(* IEC 61131-3 sources: POMIRTS_lab3/AS/Library_2/MTWinder/V1.00.3, 3 files *)

(* ---- MTWinder.typ ---- *)
TYPE
	MTWinderAxisControllerIntType : 	STRUCT  (*Data for internal use.*)
		CycleTime : REAL; (*Task cycle time. Unit: [s].*)
		Configuration : MTWinderConfigurationType; (*Data for internal use.*)
		Parameters : MTWinderAxisControllerType; (*Data for internal use.*)
		ParametersValid : BOOL; (*Data for internal use.*)
		UpdateOld : BOOL; (*Data for internal use.*)
		StartSynchronizationOld : BOOL; (*Data for internal use.*)
		StopSynchronizationOld : BOOL; (*Data for internal use.*)
		EnableOld : BOOL; (*Data for internal use.*)
		Update : BOOL; (*Data for internal use.*)
		WinderRatio : LREAL; (*Data for internal use.*)
		ActualDiameter : REAL; (*Data for internal use.*)
		ActIntegrationTime : REAL; (*Data for internal use.*)
		ActProportionalGainOld : REAL; (*Data for internal use.*)
		ActProportionalGain : REAL; (*Data for internal use.*)
		ActualInertia : REAL; (*Data for internal use.*)
		RollerDensity : REAL; (*Data for internal use.*)
		StatusIDUpdate : DINT; (*Data for internal use.*)
		StatusIDCommando : DINT; (*Data for internal use.*)
		StatusIDCyclic : DINT; (*Data for internal use.*)
		InSynchronizationOld : BOOL; (*Data for internal use.*)
		SynchronizationParameters : MTWinderAxisControllerSyncType; (*Data for internal use.*)
		SetLineVelocitySampled : REAL; (*Data for internal use.*)
	END_STRUCT;
	MTWinderAxisControllerSyncEnum :
		( (*Synchronization state of the axis controller.*)
		mtWND_STATE_STOP := 0, (*Data for internal use.*)
		mtWND_STATE_RAMP_UP := 1, (*Data for internal use.*)
		mtWND_STATE_IN_SYNC := 2, (*Data for internal use.*)
		mtWND_STATE_RAMP_DOWN := 3 (*Data for internal use.*)
		);
	MTWinderAxisControllerSyncType : 	STRUCT  (*Ramp up time parameters for the synchronization.*)
		SyncState : MTWinderAxisControllerSyncEnum; (*Data for internal use.*)
		SyncLineVelocity : REAL; (*Data for internal use.*)
		SyncLineVelocityOld : REAL; (*Data for internal use.*)
		SyncLineAcceleration : REAL; (*Data for internal use.*)
		alpha : REAL; (*Data for internal use.*)
		SyncTime : REAL; (*Data for internal use.*)
	END_STRUCT;
	MTWinderAxisControllerType : 	STRUCT  (*Parameter for the winder axis.*)
		MinTorque : REAL; (*Lower limit for the motor torque preset value SetMotorTorque. Unit: [Nm]. *)
		MaxTorque : REAL; (*Upper limit for the motor torque preset value SetMotorTorque. Unit: [Nm].*)
		Interpolation : MTWinderInterpolationType; (*Parameter for interpolating the speed controller parameters of the winder axis.*)
	END_STRUCT;
	MTWinderAxisType : 	STRUCT  (*Axis parameter.*)
		LineUnits : REAL; (*Scaling of the line position. Unit: [Units/m]. *)
		WinderUnits : UDINT; (*Scaling of the winder axis. Unit: [Units].*)
		RevMotor : UDINT; (*Number of motor revolutions required for the position of the winder to increase/decrease by a number of units equal to WinderUnits. Unit: [Rev]. *)
		GearRatio : REAL; (*Gear ratio between the motor and winder (motor speed ÷ winder speed). Unit: [1]. *)
		WinderType : MTWinderTypeEnum; (*Selects whether the system is a winder or unwinder unit.*)
		ReverseWinderDirection : BOOL; (*Changes the direction of rotation for the winder axis.*)
	END_STRUCT;
	MTWinderConfigurationType : 	STRUCT  (*Configuration parameters for the winder and the motor.*)
		Geometry : MTWinderGeometryType; (*Geometric parameter of winder.*)
		Axis : MTWinderAxisType; (*Axis parameter.*)
	END_STRUCT;
	MTWinderControllerType : 	STRUCT  (*Parameter for setting the controller.*)
		PIDParameters : MTPIDParametersType; (*PID parameter.*)
		MaxLineVelocityCorrection : REAL; (*Maximum permitted correction by controller depending on the line velocity. Unit: [mm/s].*)
		MaxControlError : REAL; (*Threshold value for detecting material failure. Unit: [mm] for closed-loop dancer control, [N] for closed-loop tension control.*)
	END_STRUCT;
	MTWinderDancerControllerIntType : 	STRUCT  (*Data for internal use.*)
		CycleTime : REAL; (*Task cycle time. Unit: [s].*)
		Configuration : MTWinderConfigurationType; (*Data for internal use.*)
		Parameters : MTWinderControllerType; (*Data for internal use.*)
		ParametersValid : BOOL; (*Data for internal use.*)
		UpdateOld : BOOL; (*Data for internal use.*)
		EnableOld : BOOL; (*Data for internal use.*)
		WinderRatio : LREAL; (*Data for internal use.*)
		ActualDiameter : REAL; (*Data for internal use.*)
		MaterialBreak : BOOL; (*Data for internal use.*)
		ControlError : REAL; (*Data for internal use.*)
		ControlErrorOld : REAL; (*Data for internal use.*)
		PIDStatusID : DINT; (*Data for internal use.*)
		ProportionalPart : REAL; (*Data for internal use.*)
		IntegrationPart : REAL; (*Data for internal use.*)
		DerivativePart : REAL; (*Data for internal use.*)
		ControllerOutput : REAL; (*Data for internal use.*)
		HoldIntegration : MTPIDIntegrationEnum; (*Data for internal use.*)
		IntegrationStatus : MTPIDIntegrationEnum; (*Data for internal use.*)
		StatusIDUpdate : DINT; (*Data for internal use.*)
	END_STRUCT;
	MTWinderDiameterEstBufferParType : 	STRUCT  (*Buffer parameters for the diameter estimator.*)
		Counter : USINT; (*Data for internal use.*)
		Index : USINT; (*Data for internal use.*)
		ActDiameter : ARRAY[0..99]OF LREAL; (*Data for internal use.*)
		WinderRevolution : ARRAY[0..99]OF LREAL; (*Data for internal use.*)
	END_STRUCT;
	MTWinderDiameterEstInternalType : 	STRUCT  (*Data for internal use.*)
		CycleTime : REAL; (*Task cycle time. Unit: [s].*)
		Configuration : MTWinderConfigurationType; (*Data for internal use.*)
		Parameters : MTWinderDiameterEstType; (*Data for internal use.*)
		ParametersValid : BOOL; (*Data for internal use.*)
		UpdateOld : BOOL; (*Data for internal use.*)
		EnableOld : BOOL; (*Data for internal use.*)
		Mode : MTWinderDiameterEstModeEnum; (*Data for internal use.*)
		SetPresetDiameterOld : BOOL; (*Data for internal use.*)
		PresetDiameter : REAL; (*Data for internal use.*)
		WinderRatio : LREAL; (*Data for internal use.*)
		RollerDensity : REAL; (*Data for internal use.*)
		SetPresetDiameterMode : USINT; (*Data for internal use.*)
		ReverseWinder : SINT; (*Data for internal use.*)
		MaterialBreak : BOOL; (*Data for internal use.*)
		SystemParameters : MTWinderDiameterEstSysParType; (*Data for internal use.*)
		EstimationParameters : MTWinderDiameterEstParType; (*Data for internal use.*)
		BufferParameters : MTWinderDiameterEstBufferParType; (*Data for internal use.*)
		LQFilter : MTWinderDiameterEstLQFilterType; (*Data for internal use.*)
		ActDiameter : REAL; (*Data for internal use.*)
		AvgMaterialThickness : REAL; (*Data for internal use.*)
		MinDiameterAchieved : BOOL; (*Data for internal use.*)
		ActLinePosition : DINT; (*Data for internal use.*)
		ActLinePositionOld : DINT; (*Data for internal use.*)
		FilterWindowTime : LREAL; (*Data for internal use.*)
		RemainingRunTime : ARRAY[0..2]OF REAL; (*Data for internal use.*)
		LineVelocity : REAL; (*Data for internal use.*)
	END_STRUCT;
	MTWinderDiameterEstLQFilterType : 	STRUCT  (*Filter parameters for the diameter estimator.*)
		LQError : REAL; (*Data for internal use.*)
		LQOutputFiltered : ARRAY[0..1]OF LREAL; (*Data for internal use.*)
		LQOutput : ARRAY[0..1]OF REAL; (*Data for internal use.*)
		LQParameterVector : ARRAY[0..2]OF REAL; (*Data for internal use.*)
		UpdateFilter : BOOL; (*Data for internal use.*)
		ResetFilter : BOOL; (*Data for internal use.*)
		InitFilter : BOOL; (*Data for internal use.*)
		NumberOfDataVector : UDINT; (*Data for internal use.*)
		BVector : ARRAY[0..1]OF DINT; (*Data for internal use.*)
		XVector : ARRAY[0..1]OF LREAL; (*Data for internal use.*)
	END_STRUCT;
	MTWinderDiameterEstModeEnum :
		( (*Diameter estimation mode.*)
		mtWND_NO_ESTIMATION := 0, (*Disables the diameter estimation.*)
		mtWND_POSITION_BASED := 1, (*Cyclic diameter estimation based on differences in position.*)
		mtWND_VELOCITY_INTEGRATION_BASED := 2 (*Cyclic diameter estimation based on integrated speeds.*)
		);
	MTWinderDiameterEstParType : 	STRUCT  (*Estimation parameters for the diameter estimator.*)
		ActDiameter : LREAL; (*Data for internal use.*)
		ActDiameterOld : REAL; (*Data for internal use.*)
		ActDiameterCorrect : REAL; (*Data for internal use.*)
		ActDiameterStart : REAL; (*Data for internal use.*)
		StartEstimation : BOOL; (*Data for internal use.*)
		StartLinePosition : DINT; (*Data for internal use.*)
		StartWinderPosition : DINT; (*Data for internal use.*)
		StartDancerPosition : REAL; (*Data for internal use.*)
		LinePositionIntegration : LREAL; (*Data for internal use.*)
		WinderPositionIntegration : LREAL; (*Data for internal use.*)
		ActWinderRevolution : ARRAY[0..2]OF LREAL; (*Data for internal use.*)
		WinderRevolution : LREAL; (*Data for internal use.*)
		ActLinePositionOld : DINT; (*Data for internal use.*)
	END_STRUCT;
	MTWinderDiameterEstSysParType : 	STRUCT  (*System parameters for the diameter estimator.*)
		ActWinderPositionOld : DINT; (*Data for internal use.*)
		ActWinderPositionDelta : DINT; (*Data for internal use.*)
		ActWinderRevolution : LREAL; (*Data for internal use.*)
		ActMotorRevolution : ARRAY[0..1]OF UDINT; (*Data for internal use.*)
	END_STRUCT;
	MTWinderDiameterEstType : 	STRUCT  (*Parameter for diameter estimation.*)
		CyclicEstimationWindow : UDINT; (*Duration of the cyclic estimation window for estimating the diameter. Unit: [Units].*)
		FilterWindow : UDINT; (*Position-related filter constant for the filter. Unit: [Units].*)
		MaterialBreakThreshold : REAL; (*Window for detecting material failure. Unit: [mm].*)
	END_STRUCT;
	MTWinderGeometryType : 	STRUCT  (*Geometric parameter of winder.*)
		WinderWidth : REAL; (*Width of the winder. Unit: [mm]. *)
		MaterialThickness : REAL; (*Material thickness or diameter (e.g. of the wire). Unit: [µm]. *)
		MaxDiameter : REAL; (*Maximum winder diameter. Unit: [mm]. *)
		MinDiameter : REAL; (*Minimum winder diameter. Unit: [mm].*)
		MinInertia : REAL; (*Moment of inertia of the winder at diameter MinDiameter. Unit: [kgm˛]. *)
		TestDiameter : REAL; (*Winder diameter between the minimum and maximum diameter at which the TestInertia or TestProportionalGain and TestIntegrationTime are determined. This diameter should be as large as possible. Unit: [mm].*)
		TestInertia : REAL; (*Moment of inertia of the winder at diameter TestDiameter. Unit: [kgm˛]. *)
	END_STRUCT;
	MTWinderInterpolationType : 	STRUCT  (*Parameter for interpolating the speed controller parameters of the winder axis.*)
		MinProportionalGain : REAL; (*Proportional gain of speed controller at minimum diameter MinDiameter. Unit: [As].*)
		TestProportionalGain : REAL; (*Proportional gain of speed controller at diameter TestDiameter. Unit: [As].*)
		MinIntegrationTime : REAL; (*Integration time of speed controller at minimum diameter. Unit: [s].*)
		TestIntegrationTime : REAL; (*Integration time of speed controller at diameter TestDiameter. Unit: [s].*)
	END_STRUCT;
	MTWinderModelTypeEnum :
		( (*Model for the winder application.*)
		mtWND_DANCER := 0, (*Uses the simulation model for dancer control.*)
		mtWND_TENSION_CLOSED_LOOP := 1, (*Uses the simulation model for closed-loop tension control.*)
		mtWND_TENSION_OPEN_LOOP := 2 (*Uses the simulation model for open-loop tension control.*)
		);
	MTWinderSimMaterialParType : 	STRUCT  (*Simulation model material parameters.*)
		RollerDensity : REAL; (*Roller density [kg/mł].*)
		ElasticityConstant : REAL; (*Elacticity constant [N/mm˛].*)
		Elongation : REAL; (*Elongation [N/m˛].*)
		Material : USINT; (*Plastic = 0. Paper = 1.*)
	END_STRUCT;
	MTWinderSimSystemParType : 	STRUCT  (*Simulation model system parameters.*)
		LinePosition : LREAL; (*Actual line position, [m]*)
		LineVelocity : LREAL; (*Actual line velocity, [m/s]*)
		IntegratorState : LREAL; (*Integrator state.*)
		MaterialTension : ARRAY[0..2]OF LREAL; (*Material tension [N].*)
		DancerArmPosition : ARRAY[0..2]OF LREAL; (*Dancer arm position [rad].*)
		DancerArmVelocity : ARRAY[0..2]OF LREAL; (*Dancer arm velocity [rad/s].*)
		WinderRollerPosition : ARRAY[0..2]OF LREAL; (*Winder roller position [rad].*)
		WinderRollerVelocity : ARRAY[0..2]OF LREAL; (*Winder roller velocity [rad/s].*)
		UnwoundMaterialLength : ARRAY[0..2]OF LREAL; (*Unwound material length [mm].*)
	END_STRUCT;
	MTWinderSimulationModelIntType : 	STRUCT  (*Data for internal use.*)
		CycleTime : REAL; (*Task cycle time. Unit: [s].*)
		Configuration : MTWinderConfigurationType; (*Data for internal use.*)
		Parameters : MTWinderSimulationModelType; (*Data for internal use.*)
		SystemParameters : MTWinderSimSystemParType; (*Data for internal use.*)
		MaterialParameters : MTWinderSimMaterialParType; (*Data for internal use.*)
		ParametersValid : BOOL; (*Data for internal use.*)
		UpdateOld : BOOL; (*Data for internal use.*)
		EnableOld : BOOL; (*Data for internal use.*)
		ActualDiameter : REAL; (*Data for internal use.*)
		InitSpeedControllerOld : REAL; (*Data for internal use.*)
		ActProportionalGain : REAL; (*Data for internal use.*)
		ActIntegrationTime : REAL; (*Data for internal use.*)
		MaterialBreak : BOOL; (*Data for internal use.*)
		ModelType : MTWinderModelTypeEnum; (*Data for internal use.*)
		TorqueMode : MTWinderTorqueModeEnum; (*Data for internal use.*)
		Update : BOOL; (*Data for internal use.*)
		InhibitUpdate : BOOL; (*Data for internal use.*)
	END_STRUCT;
	MTWinderSimulationModelType : 	STRUCT  (*Parameter for the simulation model.*)
		MaterialLength : REAL; (*Material length between the unwinder and infeed or between the outfeed and winder. Unit: [mm]. *)
		StartDiameter : REAL; (*Winder diameter used to start the simulation. Unit: [mm]. *)
		MaxDancerPosition : REAL; (*Maximum position of the dancer arm. Unit: [mm]. *)
		DancerLength : REAL; (*Length of the dancer arm. Unit: [mm]. *)
		DancerInertia : REAL; (*Moment of inertia of the dancer. Unit: [kgm˛]. *)
		SpeedTorqueFactor : REAL; (*Friction coefficient for the winder proportional to the velocity. Unit: [Nms]. *)
		TorqueConstant : REAL; (*Torque constant of the motor from the winder Unit: [Nm/A]. *)
		Noise : BOOL; (*Enables noise for the ActLinePosition, ActLineVelocity, ActWinderPosition, ActWinderVelocity, ActDancerPosition and ActMaterialTension outputs.*)
	END_STRUCT;
	MTWinderTaperTensionInternalType : 	STRUCT  (*Data for internal use.*)
		CycleTime : REAL; (*Task cycle time. Unit: [s].*)
		Configuration : MTWinderConfigurationType; (*Data for internal use.*)
		Parameters : MTWinderTaperTensionType; (*Data for internal use.*)
		ParametersValid : BOOL; (*Data for internal use.*)
		UpdateOld : BOOL; (*Data for internal use.*)
		EnableOld : BOOL; (*Data for internal use.*)
		ActualDiameter : REAL; (*Data for internal use.*)
		StartMotorTorque : REAL; (*Data for internal use.*)
		MaxMotorTorque : REAL; (*Data for internal use.*)
		MinMotorTorque : REAL; (*Data for internal use.*)
		SetMotorTorque : REAL; (*Data for internal use.*)
		StatusIDUpdate : DINT; (*Data for internal use.*)
	END_STRUCT;
	MTWinderTaperTensionModeEnum :
		( (*Tension curve mode.*)
		mtWND_LINEAR_DECREASE_TENSION := 0, (*Linear reduction of the tension.*)
		mtWND_LINEAR_DECREASE_TORQUE := 1 (*Linear reduction of the torque.*)
		);
	MTWinderTaperTensionType : 	STRUCT  (*Parameter for determining the tension profile.*)
		StartDiameter : REAL; (*Tension is reduced beginning with this diameter. Unit: [mm].*)
		MaxMaterialTension : REAL; (*Maximum tension. Unit: [N].*)
		MinMaterialTension : REAL; (*Minimum tension. Unit: [N].*)
		Mode : MTWinderTaperTensionModeEnum; (*Tension curve mode.*)
	END_STRUCT;
	MTWinderTensionControllerIntType : 	STRUCT  (*Data for internal use.*)
		CycleTime : REAL; (*Task cycle time. Unit: [s].*)
		Configuration : MTWinderConfigurationType; (*Data for internal use.*)
		Parameters : MTWinderControllerType; (*Data for internal use.*)
		ParametersValid : BOOL; (*Data for internal use.*)
		UpdateOld : BOOL; (*Data for internal use.*)
		EnableOld : BOOL; (*Data for internal use.*)
		WinderRatio : LREAL; (*Data for internal use.*)
		ActualDiameter : REAL; (*Data for internal use.*)
		MaterialBreak : BOOL; (*Data for internal use.*)
		ControlError : REAL; (*Data for internal use.*)
		ControlErrorOld : REAL; (*Data for internal use.*)
		PIDStatusID : DINT; (*Data for internal use.*)
		ProportionalPart : REAL; (*Data for internal use.*)
		IntegrationPart : REAL; (*Data for internal use.*)
		DerivativePart : REAL; (*Data for internal use.*)
		ControllerOutput : REAL; (*Data for internal use.*)
		HoldIntegration : MTPIDIntegrationEnum; (*Data for internal use.*)
		IntegrationStatus : MTPIDIntegrationEnum; (*Data for internal use.*)
		StatusIDUpdate : DINT; (*Data for internal use.*)
	END_STRUCT;
	MTWinderTorqueModeEnum :
		( (*Specifies how the value of the SetMotorTorque input is used.*)
		mtWND_TORQUE_LIMIT := 40, (*Uses SetMotorTorque for torque limiting.*)
		mtWND_TORQUE_FF := 32 (*Uses SetMotorTorque for feed-forward torque control.*)
		);
	MTWinderTypeEnum :
		( (*Selects whether the system is a winder or unwinder unit.*)
		mtWND_REWIND := -1, (*Winder used for winding.*)
		mtWND_UNWIND := +1 (*Winder used for unwinding.*)
		);
END_TYPE

(* ---- MTWinder.var ---- *)
(*Errors: Common*)
VAR CONSTANT
	mtWND_ERR_GEO_PAR_INVALID : DINT := -1058007184; (*Geometric parameter set for winder is invalid.*)
	mtWND_ERR_AXIS_PAR_INVALID : DINT := -1058007183; (*Axis parameter set for winder is invalid.*)
	mtWND_ERR_MATERIAL_BREAK : DINT := -1058007181; (*Material breakage detected.*)
	mtWND_ERR_ACT_DIAMETER_INVALID : DINT := -1058007167; (*Actual diameter for winder is invalid.*)
END_VAR
(*Warnings: Common*)
VAR CONSTANT
	mtWND_WRN_GEO_PAR_INVALID : DINT := -2131749008; (*Geometric parameter set for winder is invalid.*)
	mtWND_WRN_AXIS_PAR_INVALID : DINT := -2131749007; (*Axis parameter set for winder is invalid.*)
	mtWND_WRN_ACT_DIAMETER_INVALID : DINT := -2131748994; (*Actual diameter for winder is invalid.*)
END_VAR
(*Errors: MTWinderAxisController*)
VAR CONSTANT
	mtWND_ERR_TORQUE_LIMITS_INVALID : DINT := -1058007173; (*Torque limits set for winder are invalid.*)
	mtWND_ERR_INTERPOL_PAR_INVALID : DINT := -1058007172; (*Interpolation parameters are invalid.*)
	mtWND_ERR_SET_MAT_TENSION_NEG : DINT := -1058007169; (*Set material tension is negative.*)
END_VAR
(*Warnings: MTWinderAxisController*)
VAR CONSTANT
	mtWND_WRN_TORQUE_LIMITS_INVALID : DINT := -2131749001; (*Torque limits set for winder are invalid.*)
	mtWND_WRN_INTERPOL_PAR_INVALID : DINT := -2131749000; (*Interpolation parameters are invalid.*)
	mtWND_WRN_SYNC_TIME_NEGATIVE : DINT := -2131748996; (*Synchronization time for winder is invalid.*)
END_VAR
(*Errors: MTWinderDancerController and MTWinderTensionController*)
VAR CONSTANT
	mtWND_ERR_MAX_CONTROL_ERROR_NEG : DINT := -1058007176; (*Max control error for material detection is negative.*)
	mtWND_ERR_LINE_VEL_CORRECTION : DINT := -1058007166; (*Maximum line velocity correction is negative or equal to 0.*)
END_VAR
(*Warnings: MTWinderDancerController and MTWinderTensionController*)
VAR CONSTANT
	mtWND_WRN_MAX_CONTROL_ERROR_NEG : DINT := -2131749004; (*Max control error for material detection is negative.*)
	mtWND_WRN_LINE_VEL_CORRECTION : DINT := -2131748993; (*Maximum line velocity correction is negative or equal to 0.*)
END_VAR
(*Errors: MTWinderDiameterEstimator*)
VAR CONSTANT
	mtWND_ERR_DIAMETER_EST_MODE : DINT := -1058007177; (*Mode for the diameter estimator is invalid.*)
	mtWND_ERR_CYCLIC_EST_WINDOW : DINT := -1058007175; (*Cyclic estimation window for the diameter estimation is invalid.*)
	mtWND_ERR_MAT_BREAK_THRESHOLD : DINT := -1058007168; (*Threshold for material break detection is invalid.*)
END_VAR
(*Warnings: MTWinderDiameterEstimator*)
VAR CONSTANT
	mtWND_WRN_DIAMETER_EST_MODE : DINT := -2131749005; (*Mode for the diameter estimator is invalid.*)
	mtWND_WRN_CYCLIC_EST_WINDOW : DINT := -2131749003; (*Cyclic estimation window for the diameter estimator is invalid.*)
	mtWND_WRN_MIN_DIAMETER_REACHED : DINT := -2131749002; (*The diameter estimator has reached the minimum diameter.*)
	mtWND_WRN_MAT_BREAK_THRESHOLD : DINT := -2131748995; (*Threshold for material break detection is invalid.*)
	mtWND_WRN_PRESET_DIAMETER : DINT := -2131748990; (*Preset diameter for the diameter estimator is invalid.*)
END_VAR
(*Errors: MTWinderSimulationModel*)
VAR CONSTANT
	mtWND_ERR_SIM_PAR_INVALID : DINT := -1058007182; (*Simulation parameter set for winder is invalid.*)
	mtWND_ERR_MODEL_TYPE_INVALID : DINT := -1058007180; (*Type of model is invalid.*)
	mtWND_ERR_TORQUE_MODE_INVALID : DINT := -1058007179; (*Torque mode of model is invalid.*)
	mtWND_ERR_MODEL_TORQUE_INVALID : DINT := -1058007178; (*Torque mode for selected model type is invalid.*)
END_VAR
(*Warnings: MTWinderSimulationModel*)
VAR CONSTANT
	mtWND_WRN_SIM_PAR_INVALID : DINT := -2131749006; (*Simulation parameter set for winder is invalid.*)
END_VAR
(*Errors: MTWinderTaperTension*)
VAR CONSTANT
	mtWND_ERR_START_DIAMETER_INVALID : DINT := -1058007171; (*Start diameter for winder is invalid.*)
	mtWND_ERR_MATERIAL_TENSION_LIMIT : DINT := -1058007165; (*The maximum and the minimum material tension is invalid.*)
	mtWND_ERR_TAPER_TENSION_MODE : DINT := -1058007164; (*Mode for the taper tension is invalid.*)
END_VAR
(*Warnings: MTWinderTaperTension*)
VAR CONSTANT
	mtWND_WRN_START_DIAMETER_INVALID : DINT := -2131748999; (*Start diameter for winder is invalid.*)
	mtWND_WRN_MATERIAL_TENSION_LIMIT : DINT := -2131748992; (*The maximum and the minimum material tension is invalid.*)
	mtWND_WRN_TAPER_TENSION_MODE : DINT := -2131748991; (*Mode for the taper tension is invalid.*)
END_VAR

(* ---- MTWinder.fun ---- *)
{REDUND_OK} FUNCTION_BLOCK MTWinderAxisController (*This function block implements feed-forward control for velocity and torque that is dependent on the winder diameter.*)
	VAR_INPUT
		Enable : BOOL; (*Enables/Disables the function block.*) (* *) (*#PAR#*)
		Configuration : MTWinderConfigurationType; (*Parameter for configuring the winder.*) (* *) (*#PAR#*)
		Parameters : MTWinderAxisControllerType; (*Parameter for the winder axis.*) (* *) (*#PAR#*)
		Update : BOOL; (*Parameters are updated on a rising edge.*) (* *) (*#PAR#*)
		SetLineVelocity : REAL; (*Line velocity. Unit: [Units/s]*) (* *) (*#CYC#*)
		ActDiameter : REAL; (*Winder diameter. Unit: [mm]. *) (* *) (*#CYC#*)
		SetMaterialTension : REAL; (*Set value for material tension Unit: [N].*) (* *) (*#CYC#*)
		SynchronizationTime : REAL; (*Synchronization time. Unit: [s]. *) (* *) (*#CMD##OPT#*)
		StartSynchronization : BOOL; (*A rising edge starts a new synchronization of the winder axis (in SynchronizationTime) to the predefined line velocity.*) (* *) (*#CMD##OPT#*)
		StopSynchronization : BOOL; (*A rising edge brakes the movement of the winder axis (in SynchronizationTime).*) (* *) (*#CMD##OPT#*)
	END_VAR
	VAR_OUTPUT
		Busy : BOOL; (*The function block is not yet completed. *) (* *) (*#PAR#*)
		Active : BOOL; (*The function block is active.*) (* *) (*#PAR#*)
		Error : BOOL; (*Indicates an error.*) (* *) (*#PAR#*)
		StatusID : DINT; (*Status information.*) (* *) (*#PAR#*)
		UpdateDone : BOOL; (*Update completed.*) (* *) (*#PAR#*)
		SetWinderVelocity : REAL; (*Setpoint for the winder velocity. Unit: [Units/s].*) (* *) (*#CMD##OPT#*)
		SetMotorTorque : REAL; (*Setpoint for the motor torque. Unit: [Nm].*) (* *) (*#CYC#*)
		ActProportionalGain : REAL; (*Interpolated proportional gain of the speed controller. Unit: [As].*) (* *) (*#CYC#*)
		ActIntegrationTime : REAL; (*Interpolated integration time constant of the speed controller. Unit: [s].*) (* *) (*#CYC#*)
		InitSpeedController : BOOL; (*Generates a rising edge when initialization of the speed controller is required.*) (* *) (*#CYC#*)
		ActInertia : REAL; (*Moment of inertia of the winder/unwinder for the current diameter. Unit: [kgm˛]. *)
		InSynchronization : BOOL; (*Winder and line velocity synchronized.*) (* *) (*#CYC#*)
	END_VAR
	VAR
		Internal : MTWinderAxisControllerIntType; (*Data for internal use.*)
	END_VAR
END_FUNCTION_BLOCK

{REDUND_OK} FUNCTION_BLOCK MTWinderDancerController (*This function block implements a closed-loop controller optimized for dancer control.*)
	VAR_INPUT
		Enable : BOOL; (*Enables/Disables the function block.*) (* *) (*#PAR#*)
		Configuration : MTWinderConfigurationType; (*Parameter for configuring the winder.*) (* *) (*#PAR#*)
		Parameters : MTWinderControllerType; (*Parameter for setting the controller.*) (* *) (*#PAR#*)
		Update : BOOL; (*Parameters are updated on a rising edge.*) (* *) (*#PAR#*)
		SetDancerPosition : REAL; (*Setpoint for the dancer position. Unit: [mm].*) (* *) (*#CYC#*)
		ActDancerPosition : REAL; (*Actual value for the dancer position. Unit: [mm].*) (* *) (*#CYC#*)
		ActDiameter : REAL; (*Current winder diameter. Unit: [mm].*) (* *) (*#CYC#*)
		Hold : BOOL; (*Freezes the function block.*) (* *) (*#CMD##OPT#*)
	END_VAR
	VAR_OUTPUT
		Active : BOOL; (*The function block is active.*) (* *) (*#PAR#*)
		Error : BOOL; (*Indicates an error.*) (* *) (*#PAR#*)
		StatusID : DINT; (*Status information.*) (* *) (*#PAR#*)
		UpdateDone : BOOL; (*Update completed.*) (* *) (*#PAR#*)
		VelocityCorrection : REAL; (*Calculated correction velocity for the winder axis. Unit: [Units/s].*) (* *) (*#CYC#*)
		MaterialBreak : BOOL; (*Indicates material failure.*) (* *) (*#CMD##OPT#*)
	END_VAR
	VAR
		Internal : MTWinderDancerControllerIntType; (*Data for internal use.*)
	END_VAR
END_FUNCTION_BLOCK

{REDUND_OK} FUNCTION_BLOCK MTWinderDiameterEstimator (*This function block implements diameter estimation for winder and unwinder systems.*)
	VAR_INPUT
		Enable : BOOL; (*Enables/Disables the function block.*) (* *) (*#PAR#*)
		Configuration : MTWinderConfigurationType; (*Parameter for configuring the winder.*) (* *) (*#PAR#*)
		Parameters : MTWinderDiameterEstType; (*Parameter for diameter estimation.*) (* *) (*#PAR#*)
		Mode : MTWinderDiameterEstModeEnum; (*Diameter estimation mode.*)
		Update : BOOL; (*Parameters are updated on a rising edge.*) (* *) (*#PAR#*)
		ActLinePosition : DINT; (*Measured actual position of the line. Unit: [Units].*)
		ActLineVelocity : REAL; (*Measured actual velocity of the line. Unit: [Units/s].*)
		ActWinderPosition : DINT; (*Measured actual position of the winder axis. Unit: [Units].*)
		ActWinderVelocity : REAL; (*Measured actual velocity of the winder. Unit: [Units/s].*)
		ActDancerPosition : REAL; (*Actual value for the dancer position. Unit: [mm].*)
		PresetDiameter : REAL; (*Preset value for the winder diameter. Unit: [mm]. *)
		SetPresetDiameter : BOOL; (*A rising edge sets ActDiameter = PresetDiameter.*)
		Hold : BOOL; (*Freezes the function block.*)
	END_VAR
	VAR_OUTPUT
		Active : BOOL; (*The function block is active.*) (* *) (*#PAR#*)
		Error : BOOL; (*Indicates an error.*) (* *) (*#PAR#*)
		StatusID : DINT; (*Status information.*) (* *) (*#PAR#*)
		UpdateDone : BOOL; (*Update completed.*) (* *) (*#PAR#*)
		ActDiameter : REAL; (*Estimated winder diameter. Unit: [mm]. *)
		AvgMaterialThickness : REAL; (*Average material thickness. Unit: [µm]. *)
		AvgMaterialDensity : REAL; (*Average material density. Unit: [kg/mł]. *)
		ProcessedMaterial : REAL; (*Material being processed on the winder. Unit: [m].*)
		RemainingRunTime : REAL; (*Time remaining until the rest of the material is wound/unwound. Unit: [s].*)
		MaterialBreak : BOOL; (*Indicates material failure.*)
	END_VAR
	VAR
		Internal : MTWinderDiameterEstInternalType; (*Data for internal use.*)
	END_VAR
END_FUNCTION_BLOCK

{REDUND_OK} FUNCTION_BLOCK MTWinderSimulationModel (*This function block implements a simulation model for winder and unwinder systems.*)
	VAR_INPUT
		Enable : BOOL; (*Enables/Disables the function block.*) (* *) (*#PAR#*)
		Configuration : MTWinderConfigurationType; (*Parameter for configuring the winder.*) (* *) (*#PAR#*)
		Parameters : MTWinderSimulationModelType; (*Parameter for the simulation model.*) (* *) (*#PAR#*)
		Update : BOOL; (*Parameters are updated on a rising edge.*) (* *) (*#PAR#*)
		ModelType : MTWinderModelTypeEnum; (*Model for the winder application.*) (* *) (*#PAR#*)
		TorqueMode : MTWinderTorqueModeEnum; (*Specifies how the value of the SetMotorTorque input is used.*) (* *) (*#PAR#*)
		SetLineVelocity : REAL; (*Preset value for the line velocity. Unit: [m/min].*) (* *) (*#CYC#*)
		SetWinderVelocity : REAL; (*Velocity setpoint of the winder. Unit: [Units/s]*) (* *) (*#CYC#*)
		WinderVelocityCorrection : REAL; (*Correction velocity of the winder. Unit: [Units/s]*) (* *) (*#CYC#*)
		SetMotorTorque : REAL; (*Torque for feed-forward control or torque limiting. Unit: [Nm].*) (* *) (*#CYC#*)
		SetDancerTorque : REAL; (*Torque applied to the dancer arm. Unit: [Nm]. *) (* *) (*#CYC#*)
		ActProportionalGain : REAL; (*Proportional gain of the speed controller. Unit: [As].*) (* *) (*#CMD##OPT#*)
		ActIntegrationTime : REAL; (*Integral action time of the speed controller. Unit: [s].*) (* *) (*#CMD##OPT#*)
		InitSpeedController : BOOL; (*The parameters ActProportionalGain and ActIntegrationTime are updated on a rising edge of an input.*) (* *) (*#CMD##OPT#*)
		MaterialBreak : BOOL; (*A rising edge simulates material failure. *) (* *) (*#CMD##OPT#*)
	END_VAR
	VAR_OUTPUT
		Active : BOOL; (*Function block is active.*) (* *) (*#PAR#*)
		Error : BOOL; (*Indicates an error.*) (* *) (*#PAR#*)
		StatusID : DINT; (*Status information.*) (* *) (*#PAR#*)
		UpdateDone : BOOL; (*Update completed.*) (* *) (*#PAR#*)
		ActLinePosition : DINT; (*Actual position of the line. Unit: [Units].*) (* *) (*#CYC#*)
		ActLineVelocity : REAL; (*Actual speed of the line. Unit: [Units/s].*) (* *) (*#CYC#*)
		ActWinderPosition : DINT; (*Actual position of the winder. Unit: [Units].*) (* *) (*#CYC#*)
		ActWinderVelocity : REAL; (*Actual winder velocity. Units: [Units/s].*) (* *) (*#CYC#*)
		ActDancerPosition : REAL; (*Actual position of the dancer. Unit: [mm]. *) (* *) (*#CYC#*)
		ActDiameter : REAL; (*Actual diameter of the winder. Unit: [mm]. *) (* *) (*#CYC#*)
		ActMaterialTension : REAL; (*Actual tension of the material. Unit: [N].*) (* *) (*#CYC#*)
		ActMotorTorque : REAL; (*Actual torque of the winder motor. Unit: [Nm]. *) (* *) (*#CYC#*)
	END_VAR
	VAR
		Internal : MTWinderSimulationModelIntType; (*Data for internal use.*)
	END_VAR
END_FUNCTION_BLOCK

{REDUND_OK} FUNCTION_BLOCK MTWinderTaperTension (*This function block generates a tension curve in relation to the diameter. *)
	VAR_INPUT
		Enable : BOOL; (*Enables/Disables the function block.*) (* *) (*#PAR#*)
		Configuration : MTWinderConfigurationType; (*Configuration parameters for the winder and the motor.*) (* *) (*#PAR#*)
		Parameters : MTWinderTaperTensionType; (*Parameter for determining the tension profile.*) (* *) (*#PAR#*)
		Update : BOOL; (*Parameters are updated on a rising edge.*) (* *) (*#PAR#*)
		ActDiameter : REAL; (*Current winder diameter. Unit: [mm].*) (* *) (*#CMD##OPT#*)
	END_VAR
	VAR_OUTPUT
		Active : BOOL; (*The function block is active. *) (* *) (*#PAR#*)
		Error : BOOL; (*Indicates an error.*) (* *) (*#PAR#*)
		StatusID : DINT; (*Status information.*) (* *) (*#PAR#*)
		UpdateDone : BOOL; (*Update completed.*) (* *) (*#PAR#*)
		SetMaterialTension : REAL; (*Setpoint for the tension. Unit: [N]*) (* *) (*#CYC#*)
	END_VAR
	VAR
		Internal : MTWinderTaperTensionInternalType; (*Data for internal use.*)
	END_VAR
END_FUNCTION_BLOCK

{REDUND_OK} FUNCTION_BLOCK MTWinderTensionController (*This function block implements a closed-loop tension controller.*)
	VAR_INPUT
		Enable : BOOL; (*Enables/Disables the function block.*) (* *) (*#PAR#*)
		Configuration : MTWinderConfigurationType; (*Parameter for configuring the winder.*) (* *) (*#PAR#*)
		Parameters : MTWinderControllerType; (*Parameter for setting the controller.*) (* *) (*#PAR#*)
		Update : BOOL; (*Parameters are updated on a rising edge.*) (* *) (*#PAR#*)
		SetMaterialTension : REAL; (*Setpoint for the tension. Unit: [N]*) (* *) (*#CYC#*)
		ActMaterialTension : REAL; (*Current tension. Unit: [N]*) (* *) (*#CYC#*)
		ActDiameter : REAL; (*Current winder diameter. Unit: [mm].*) (* *) (*#CYC#*)
		Hold : BOOL; (*Freezes the function block.*) (* *) (*#CMD##OPT#*)
	END_VAR
	VAR_OUTPUT
		Active : BOOL; (*Function block is active.*) (* *) (*#PAR#*)
		Error : BOOL; (*Indicates an error.*) (* *) (*#PAR#*)
		StatusID : DINT; (*Status information.*) (* *) (*#PAR#*)
		UpdateDone : BOOL; (*Update completed.*) (* *) (*#PAR#*)
		VelocityCorrection : REAL; (*Calculated correction velocity for the winder axis. Unit: [units/s]*) (* *) (*#CYC#*)
		MaterialBreak : BOOL; (*Indicates material failure.*) (* *) (*#CMD##OPT#*)
	END_VAR
	VAR
		Internal : MTWinderTensionControllerIntType; (*Data for internal use.*)
	END_VAR
END_FUNCTION_BLOCK
